(* IEC 61131-3 sources: AXOpen/src/components.keyence.vision/ctrl/src/Axo_IV3/TypesStructuresAndEnums, 15 files *)

(* ---- Axo_IV3_CommandControl.st ---- *)
NAMESPACE AXOpen.Components.Keyence.Vision
    {S7.extern=ReadWrite}
    {#ix-attr:[Container(Layout.Stack)]}
    CLASS PUBLIC Axo_IV3_CommandControl
        VAR PUBLIC
            {#ix-set:AttributeName = "<#Trigger request#>"}
            TriggerRequest                              : BOOL;                         //  QB0.0
            {#ix-set:AttributeName = "<#Master registration request#>"}
            MasterRegistrationRequest                   : BOOL;                         //  QB0.1
            {#ix-set:AttributeName = "<#Program switching request#>"}
            ProgramSwitchingRequest                     : BOOL;                         //  QB0.2
            {#ix-set:AttributeName = "<#Warning clear request#>"}
            WarningClearRequest                         : BOOL;                         //  QB0.3
            {#ix-set:AttributeName = "<#Statistics reset request#>"}
            StatisticsResetRequest                      : BOOL;                         //  QB0.4
            {#ix-set:AttributeName = "<#Buffer clear request#>"}
            BufferClearRequest                          : BOOL;                         //  QB0.5
            {#ix-set:AttributeName = "<#SD card saving stop request#>"}
            SdCardSavingStopRequest                     : BOOL;                         //  QB0.6
            {#ix-set:AttributeName = "<#Setting value change request#>"}
            SettingValueChangeRequest                   : BOOL;                         //  QB0.7
            {#ix-set:AttributeName = "<#Result acquisition complete notification#>"}
            ResultAcquisitionCompleteNotification       : BOOL;                         //  QB2.0
            {#ix-set:AttributeName = "<#Program number#>"}
            ProgramNo                                   : UINT;                         //  QW4
            {#ix-set:AttributeName = "<#Function 1: Limit set.no.(no OCR)/Master text set.no.(OCR)/FTP/SD-saved set.no.(FTP client/SD card saving function)#>"}
            Function_1                                  : WORD;                         //  QW6
            {#ix-set:AttributeName = "<#Function 2: Limit set.no.(no OCR)/Master text/number of letters(OCR)/FTP/SD-saving settings(FTP client/SD card saving function)#>"}
            Function_2                                  : DWORD;                        //  QD8
        END_VAR
    END_CLASS
END_NAMESPACE

(* ---- Axo_IV3_CommandStatusBits.st ---- *)
NAMESPACE AXOpen.Components.Keyence.Vision
    {S7.extern=ReadWrite}
    {#ix-attr:[Container(Layout.Wrap)]}
    CLASS PUBLIC Axo_IV3_CommandStatusBits
        VAR PUBLIC
            {#ix-attr:[Container(Layout.Stack)]}
            {#ix-attr:[Group(GroupLayout.GroupBox)]}
            {#ix-set:AttributeName = "<#Trigger response#>"}
            TriggerResponse : BOOL;                                                             // IB0.0
            {#ix-set:AttributeName = "<#Master registration response#>"}
            MasterRegistrationResponse : BOOL;                                                  // IB0.1
            {#ix-set:AttributeName = "<#Program switching response#>"}
            ProgramSwitchingResponse : BOOL;                                                    // IB0.2
            {#ix-set:AttributeName = "<#Warning clear response#>"}
            WarningClearResponse : BOOL;                                                        // IB0.3
            {#ix-set:AttributeName = "<#Statistics reset response#>"}
            StatisticsResetResponse : BOOL;                                                     // IB0.4
            {#ix-set:AttributeName = "<#Buffer clear response#>"}
            BufferClearResponse : BOOL;                                                         // IB0.5
            {#ix-set:AttributeName = "<#SD card saving stop response#>"}
            SdCardSavingStopResponse : BOOL;                                                    // IB0.6
            {#ix-set:AttributeName = "<#Setting value change response#>"}
            SettingValueChangeResponse : BOOL;                                                  // IB0.7

            {#ix-attr:[Container(Layout.Stack)]}
            {#ix-attr:[Group(GroupLayout.GroupBox)]}
            {#ix-set:AttributeName = "<#Trigger failed#>"}
            TriggerFailed : BOOL;                                                               // IB1.0
            {#ix-set:AttributeName = "<#Master registration failed#>"}
            MasterRegistrationFailed : BOOL;                                                    // IB1.1
            {#ix-set:AttributeName = "<#Program switching failed#>"}
            ProgramSwitchingFailed : BOOL;                                                      // IB1.2
                                                                                                // IB1.3
                                                                                                // IB1.4
                                                                                                // IB1.5
            {#ix-set:AttributeName = "<#SD card saving stop failed#>"}
            SdCardSavingStopFailed : BOOL;                                                      // IB1.6
            {#ix-set:AttributeName = "<#Setting value change failed#>"}
            SettingValueChangeFailed : BOOL;                                                    // IB1.7

            {#ix-attr:[Container(Layout.Stack)]}
            {#ix-attr:[Group(GroupLayout.GroupBox)]}
            {#ix-set:AttributeName = "<#Result available#>"}
            ResultAvailable : BOOL;                                                             // IB2.0
            {#ix-set:AttributeName = "<#Result update complete#>"}
            ResultUpdateComplete : BOOL;                                                        // IB2.1
            {#ix-set:AttributeName = "<#BUSY#>"}
            BUSY : BOOL;                                                                        // IB2.2
            {#ix-set:AttributeName = "<#Imaging status#>"}
            ImagingStatus : BOOL;                                                               // IB2.3
            {#ix-set:AttributeName = "<#RUN#>"}
            RUN : BOOL;                                                                         // IB2.4
            {#ix-set:AttributeName = "<#Ready#>"}
            Ready : BOOL;                                                                       // IB2.5
            {#ix-set:AttributeName = "<#Trigger ready#>"}
            TriggerReady : BOOL;                                                                // IB2.6
            {#ix-set:AttributeName = "<#SD card identification status#>"}
            SdCardIdentificationStatus : BOOL;                                                  // IB2.7

            {#ix-attr:[Container(Layout.Stack)]}
            {#ix-attr:[Group(GroupLayout.GroupBox)]}
            {#ix-set:AttributeName = "<#Sorting mode information#>"}
            SortingModeInformation : BOOL;                                                      // IB3.0
                                                                                                // IB3.1
                                                                                                // IB3.2
                                                                                                // IB3.3
            {#ix-set:AttributeName = "<#Insufficient free space on SD card#>"}
            InsufficientFreeSpaceOnSdCard : BOOL;                                               // IB3.4
            {#ix-set:AttributeName = "<#Buffer overrun#>"}
            BufferOverrun : BOOL;                                                               // IB3.5
            {#ix-set:AttributeName = "<#Warning#>"}
            Warning : BOOL;                                                                     // IB3.6
            {#ix-set:AttributeName = "<#Error#>"}
            Error : BOOL;                                                                       // IB3.7

        END_VAR
    END_CLASS
END_NAMESPACE

(* ---- Axo_IV3_Component_Status.st ---- *)
NAMESPACE AXOpen.Components.Keyence.Vision
    {S7.extern=ReadWrite}
    {#ix-attr:[Container(Layout.Stack)]}
    CLASS PUBLIC Axo_IV3_Component_Status EXTENDS AXOpen.Components.Abstractions.AxoComponent_Status
        VAR PUBLIC

        END_VAR
    END_CLASS
END_NAMESPACE

(* ---- Axo_IV3_Config.st ---- *)
NAMESPACE AXOpen.Components.Keyence.Vision
    {S7.extern=ReadWrite}
    {#ix-attr:[Container(Layout.Stack)]}
    CLASS PUBLIC Axo_IV3_Config
        VAR PUBLIC
            {#ix-set:AttributeName = "<#Info time#>"}
            InfoTime : LTIME := LT#5S;
            {#ix-set:AttributeName = "<#Error time#>"}
            ErrorTime : LTIME := LT#10S;
            {#ix-set:AttributeName = "<#Task timeout#>"}
            TaskTimeout : LTIME := LT#50S;
            {#ix-set:AttributeName = "<#Hardware IDs#>"}
            HWIDs : Axo_IV3_HWIDs;
        END_VAR
    END_CLASS
END_NAMESPACE

(* ---- Axo_IV3_Control.st ---- *)
NAMESPACE AXOpen.Components.Keyence.Vision
    {S7.extern=ReadWrite}
    {#ix-attr:[Container(Layout.Stack)]}
    CLASS PUBLIC Axo_IV3_Control
        VAR PUBLIC

        END_VAR
    END_CLASS
END_NAMESPACE

(* ---- Axo_IV3_DeviceResultBits_1.st ---- *)
NAMESPACE AXOpen.Components.Keyence.Vision
    {S7.extern=ReadWrite}
    {#ix-attr:[Container(Layout.Wrap)]}
    CLASS PUBLIC Axo_IV3_DeviceResultBits_1
        VAR PUBLIC
            {#ix-attr:[Container(Layout.Stack)]}
            {#ix-attr:[Group(GroupLayout.GroupBox)]}
            {#ix-set:AttributeName = "<#Overall judgment OK#>"}
            OverallJudgmentOK : BOOL;                                                           // IB4.0
            {#ix-set:AttributeName = "<#Position correction#>"}
            PositionCorrection : BOOL;                                                          // IB4.1
            {#ix-set:AttributeName = "<#LOGIC1#>"}
            LOGIC1 : BOOL;                                                                      // IB4.2
            {#ix-set:AttributeName = "<#LOGIC2#>"}
            LOGIC2 : BOOL;                                                                      // IB4.3
            {#ix-set:AttributeName = "<#LOGIC3#>"}
            LOGIC3 : BOOL;                                                                      // IB4.4
            {#ix-set:AttributeName = "<#LOGIC4#>"}
            LOGIC4 : BOOL;                                                                      // IB4.5
            {#ix-set:AttributeName = "<#Overall judgment NG#>"}
            OverallJudgmentNG : BOOL;                                                           // IB4.6
                                                                                                // IB4.7
            {#ix-attr:[Container(Layout.Stack)]}
            {#ix-attr:[Group(GroupLayout.GroupBox)]}
            {#ix-set:AttributeName = "<#Tool 1#>"}
            Tool_1 : BOOL;                                                                      // IB6.0
            {#ix-set:AttributeName = "<#Tool 2#>"}
            Tool_2 : BOOL;                                                                      // IB6.1
            {#ix-set:AttributeName = "<#Tool 3#>"}
            Tool_3 : BOOL;                                                                      // IB6.2
            {#ix-set:AttributeName = "<#Tool 4#>"}
            Tool_4 : BOOL;                                                                      // IB6.3
            {#ix-set:AttributeName = "<#Tool 5#>"}
            Tool_5 : BOOL;                                                                      // IB6.4
            {#ix-set:AttributeName = "<#Tool 6#>"}
            Tool_6 : BOOL;                                                                      // IB6.5
            {#ix-set:AttributeName = "<#Tool 7#>"}
            Tool_7 : BOOL;                                                                      // IB6.6
            {#ix-set:AttributeName = "<#Tool 8#>"}
            Tool_8 : BOOL;                                                                      // IB6.7
            {#ix-set:AttributeName = "<#Tool 9#>"}
            Tool_9 : BOOL;                                                                      // IB7.0
            {#ix-set:AttributeName = "<#Tool 10#>"}
            Tool_10 : BOOL;                                                                     // IB7.1
            {#ix-set:AttributeName = "<#Tool 11#>"}
            Tool_11 : BOOL;                                                                     // IB7.2
            {#ix-set:AttributeName = "<#Tool 12#>"}
            Tool_12 : BOOL;                                                                     // IB7.3
            {#ix-set:AttributeName = "<#Tool 13#>"}
            Tool_13 : BOOL;                                                                     // IB7.4
            {#ix-set:AttributeName = "<#Tool 14#>"}
            Tool_14 : BOOL;                                                                     // IB7.5
            {#ix-set:AttributeName = "<#Tool 15#>"}
            Tool_15 : BOOL;                                                                     // IB7.6
            {#ix-set:AttributeName = "<#Tool 16#>"}
            Tool_16 : BOOL;                                                                     // IB7.7
        END_VAR
    END_CLASS
END_NAMESPACE

(* ---- Axo_IV3_DeviceResultBits_2.st ---- *)
NAMESPACE AXOpen.Components.Keyence.Vision
    {S7.extern=ReadWrite}
    {#ix-attr:[Container(Layout.Wrap)]}
    CLASS PUBLIC Axo_IV3_DeviceResultBits_2
        VAR PUBLIC
            {#ix-attr:[Container(Layout.Stack)]}
            {#ix-attr:[Group(GroupLayout.GroupBox)]}
            {#ix-set:AttributeName = "<#Master number/total status product type#>"}
            MasterNumber : UINT;                                                                // IW1352

            {#ix-attr:[Container(Layout.Stack)]}
            {#ix-attr:[Group(GroupLayout.GroupBox)]}
            {#ix-set:AttributeName = "<#Tool 17#>"}
            Tool_17 : BOOL;                                                                      // IB1354.0
            {#ix-set:AttributeName = "<#Tool 18#>"}
            Tool_18 : BOOL;                                                                      // IB1354.1
            {#ix-set:AttributeName = "<#Tool 19#>"}
            Tool_19 : BOOL;                                                                      // IB1354.2
            {#ix-set:AttributeName = "<#Tool 20#>"}
            Tool_20 : BOOL;                                                                      // IB1354.3
            {#ix-set:AttributeName = "<#Tool 21#>"}
            Tool_21 : BOOL;                                                                      // IB1354.4
            {#ix-set:AttributeName = "<#Tool 22#>"}
            Tool_22 : BOOL;                                                                      // IB1354.5
            {#ix-set:AttributeName = "<#Tool 23#>"}
            Tool_23 : BOOL;                                                                      // IB1354.6
            {#ix-set:AttributeName = "<#Tool 24#>"}
            Tool_24 : BOOL;                                                                      // IB1354.7
            {#ix-set:AttributeName = "<#Tool 25#>"}
            Tool_25 : BOOL;                                                                      // IB1355.0
            {#ix-set:AttributeName = "<#Tool 26#>"}
            Tool_26 : BOOL;                                                                      // IB1355.1
            {#ix-set:AttributeName = "<#Tool 27#>"}
            Tool_27 : BOOL;                                                                      // IB1355.2
            {#ix-set:AttributeName = "<#Tool 28#>"}
            Tool_28 : BOOL;                                                                      // IB1355.3
            {#ix-set:AttributeName = "<#Tool 29#>"}
            Tool_29 : BOOL;                                                                      // IB1355.4
            {#ix-set:AttributeName = "<#Tool 30#>"}
            Tool_30 : BOOL;                                                                      // IB1355.5
            {#ix-set:AttributeName = "<#Tool 31#>"}
            Tool_31 : BOOL;                                                                      // IB1355.6
            {#ix-set:AttributeName = "<#Tool 32#>"}
            Tool_32 : BOOL;                                                                      // IB1355.7
            {#ix-set:AttributeName = "<#Tool 33#>"}
            Tool_33 : BOOL;                                                                      // IB1356.0
            {#ix-set:AttributeName = "<#Tool 34#>"}
            Tool_34 : BOOL;                                                                      // IB1356.1
            {#ix-set:AttributeName = "<#Tool 35#>"}
            Tool_35 : BOOL;                                                                      // IB1356.2
            {#ix-set:AttributeName = "<#Tool 36#>"}
            Tool_36 : BOOL;                                                                      // IB1356.3
            {#ix-set:AttributeName = "<#Tool 37#>"}
            Tool_37 : BOOL;                                                                      // IB1356.4
            {#ix-set:AttributeName = "<#Tool 38#>"}
            Tool_38 : BOOL;                                                                      // IB1356.5
            {#ix-set:AttributeName = "<#Tool 39#>"}
            Tool_39 : BOOL;                                                                      // IB1356.6
            {#ix-set:AttributeName = "<#Tool 40#>"}
            Tool_40 : BOOL;                                                                      // IB1356.7
            {#ix-set:AttributeName = "<#Tool 41#>"}
            Tool_41 : BOOL;                                                                      // IB1357.0
            {#ix-set:AttributeName = "<#Tool 42#>"}
            Tool_42 : BOOL;                                                                      // IB1357.1
            {#ix-set:AttributeName = "<#Tool 43#>"}
            Tool_43 : BOOL;                                                                      // IB1357.2
            {#ix-set:AttributeName = "<#Tool 44#>"}
            Tool_44 : BOOL;                                                                      // IB1357.3
            {#ix-set:AttributeName = "<#Tool 45#>"}
            Tool_45 : BOOL;                                                                      // IB1357.4
            {#ix-set:AttributeName = "<#Tool 46#>"}
            Tool_46 : BOOL;                                                                      // IB1357.5
            {#ix-set:AttributeName = "<#Tool 47#>"}
            Tool_47 : BOOL;                                                                      // IB1357.6
            {#ix-set:AttributeName = "<#Tool 48#>"}
            Tool_48 : BOOL;                                                                      // IB1357.7
            {#ix-set:AttributeName = "<#Tool 49#>"}
            Tool_49 : BOOL;                                                                      // IB1358.0
            {#ix-set:AttributeName = "<#Tool 50#>"}
            Tool_50 : BOOL;                                                                      // IB1358.1
            {#ix-set:AttributeName = "<#Tool 51#>"}
            Tool_51 : BOOL;                                                                      // IB1358.2
            {#ix-set:AttributeName = "<#Tool 52#>"}
            Tool_52 : BOOL;                                                                      // IB1358.3
            {#ix-set:AttributeName = "<#Tool 53#>"}
            Tool_53 : BOOL;                                                                      // IB1358.4
            {#ix-set:AttributeName = "<#Tool 54#>"}
            Tool_54 : BOOL;                                                                      // IB1358.5
            {#ix-set:AttributeName = "<#Tool 55#>"}
            Tool_55 : BOOL;                                                                      // IB1358.6
            {#ix-set:AttributeName = "<#Tool 56#>"}
            Tool_56 : BOOL;                                                                      // IB1358.7
            {#ix-set:AttributeName = "<#Tool 57#>"}
            Tool_57 : BOOL;                                                                      // IB1359.0
            {#ix-set:AttributeName = "<#Tool 58#>"}
            Tool_58 : BOOL;                                                                      // IB1359.1
            {#ix-set:AttributeName = "<#Tool 59#>"}
            Tool_59 : BOOL;                                                                      // IB1359.2
            {#ix-set:AttributeName = "<#Tool 60#>"}
            Tool_60 : BOOL;                                                                      // IB1359.3
            {#ix-set:AttributeName = "<#Tool 61#>"}
            Tool_61 : BOOL;                                                                      // IB1359.4
            {#ix-set:AttributeName = "<#Tool 62#>"}
            Tool_62 : BOOL;                                                                      // IB1359.5
            {#ix-set:AttributeName = "<#Tool 63#>"}
            Tool_63 : BOOL;                                                                      // IB1359.6
            {#ix-set:AttributeName = "<#Tool 64#>"}
            Tool_64 : BOOL;                                                                      // IB1359.7
        END_VAR
    END_CLASS
END_NAMESPACE

(* ---- Axo_IV3_DeviceStatistics.st ---- *)
NAMESPACE AXOpen.Components.Keyence.Vision
    {S7.extern=ReadWrite}
    {#ix-attr:[Container(Layout.Wrap)]}
    CLASS PUBLIC Axo_IV3_DeviceStatistics
        VAR PUBLIC
            {#ix-attr:[Container(Layout.Stack)]}
            {#ix-attr:[Group(GroupLayout.GroupBox)]}
            {#ix-set:AttributeName = "<#Processing time MAX#>"}
            ProcessingTimeMax : UINT;                                                           // IW24
            {#ix-set:AttributeName = "<#Processing time MIN#>"}
            ProcessingTimeMin : UINT;                                                           // IW26
            {#ix-set:AttributeName = "<#Processing time AVE#>"}
            ProcessingTimeAve : UINT;                                                           // IW28
                                                                                                // IW30
            {#ix-set:AttributeName = "<#Number of triggers#>"}
            NumberOfTriggers : UDINT;                                                           // ID32
            {#ix-set:AttributeName = "<#Number of OKs#>"}
            NumberOfOKs : UDINT;                                                                // ID36
            {#ix-set:AttributeName = "<#Number of NGs#>"}
            NumberOfNGs : UDINT;                                                                // ID40
            {#ix-set:AttributeName = "<#Number of trigger errors#>"}
            NumberOfTriggerErrors : UDINT;                                                      // ID44
                                                                                                // ID48
        END_VAR
    END_CLASS
END_NAMESPACE

(* ---- Axo_IV3_DeviceStatusWords.st ---- *)
NAMESPACE AXOpen.Components.Keyence.Vision
    {S7.extern=ReadWrite}
    {#ix-attr:[Container(Layout.Wrap)]}
    CLASS PUBLIC Axo_IV3_DeviceStatusWords
        VAR PUBLIC
            {#ix-attr:[Container(Layout.Stack)]}
            {#ix-attr:[Group(GroupLayout.GroupBox)]}
            {#ix-set:AttributeName = "<#Error No.#>"}
            ErrorNo : UINT;                                                                     // IW8
            {#ix-set:AttributeName = "<#Warning No.#>"}
            WarningNo : UINT;                                                                   // IW10
            {#ix-set:AttributeName = "<#Number of remaining buffers#>"}
            NumberOfRemainingBuffers : UINT;                                                    // IW12
            {#ix-set:AttributeName = "<#Checksum#>"}
            Checksum : UINT;                                                                    // IW14
            {#ix-set:AttributeName = "<#Current program No.#>"}
            CurrentProgramNo : UINT;                                                            // IW16
            {#ix-set:AttributeName = "<#Program No. during judgment#>"}
            ProgramNoDuringJudgment : UINT;                                                     // IW18
            {#ix-set:AttributeName = "<#Result No.#>"}
            ResultNo : UINT;                                                                    // IW20
            {#ix-set:AttributeName = "<#Processing time#>"}
            ProcessingTime : UINT;                                                              // IW22
        END_VAR
    END_CLASS
END_NAMESPACE

(* ---- Axo_IV3_HWIDs.st ---- *)
NAMESPACE AXOpen.Components.Keyence.Vision
   {S7.extern=ReadWrite}
	CLASS Axo_IV3_HWIDs
      VAR PUBLIC
         {#ix-set:AttributeName = "<#Hardware ID  of the device#>"}
         HW_Device              :  UINT;
         {#ix-set:AttributeName = "<#Hardware ID of the 'CommandControl' submodule#>"}
         HwID_CommandControl            :   UINT;
         {#ix-set:AttributeName = "<#Hardware ID of the 'CommandStatusBits' submodule#>"}
         HwID_CommandStatusBits            :   UINT;
         {#ix-set:AttributeName = "<#Hardware ID of the 'DeviceResultBits_1' submodule#>"}
         HwID_DeviceResultBits_1            :   UINT;
         {#ix-set:AttributeName = "<#Hardware ID of the 'DeviceStatusWords' submodule#>"}
         HwID_DeviceStatusWords            :   UINT;
         {#ix-set:AttributeName = "<#Hardware ID of the 'DeviceStatistics' submodule#>"}
         HwID_DeviceStatistics            :   UINT;
         {#ix-set:AttributeName = "<#Hardware ID of the 'PositionAdjustResult' submodule#>"}
         HwID_PositionAdjustResult            :   UINT;
         {#ix-set:AttributeName = "<#Hardware ID of the 'ToolResult_1' submodule#>"}
         HwID_ToolResult_1            :   UINT;
         {#ix-set:AttributeName = "<#Hardware ID of the 'ToolResult_2' submodule#>"}
         HwID_ToolResult_2            :   UINT;
         {#ix-set:AttributeName = "<#Hardware ID of the 'ToolResult_3' submodule#>"}
         HwID_ToolResult_3            :   UINT;
         {#ix-set:AttributeName = "<#Hardware ID of the 'ToolResult_4' submodule#>"}
         HwID_ToolResult_4            :   UINT;
         {#ix-set:AttributeName = "<#Hardware ID of the 'ToolResult_5' submodule#>"}
         HwID_ToolResult_5            :   UINT;
         {#ix-set:AttributeName = "<#Hardware ID of the 'ToolResult_6' submodule#>"}
         HwID_ToolResult_6            :   UINT;
         {#ix-set:AttributeName = "<#Hardware ID of the 'ToolResult_7' submodule#>"}
         HwID_ToolResult_7            :   UINT;
         {#ix-set:AttributeName = "<#Hardware ID of the 'ToolResult_8' submodule#>"}
         HwID_ToolResult_8            :   UINT;
         {#ix-set:AttributeName = "<#Hardware ID of the 'ToolResult_9' submodule#>"}
         HwID_ToolResult_9            :   UINT;
         {#ix-set:AttributeName = "<#Hardware ID of the 'ToolResult_10' submodule#>"}
         HwID_ToolResult_10            :   UINT;
         {#ix-set:AttributeName = "<#Hardware ID of the 'ToolResult_11' submodule#>"}
         HwID_ToolResult_11            :   UINT;
         {#ix-set:AttributeName = "<#Hardware ID of the 'ToolResult_12' submodule#>"}
         HwID_ToolResult_12            :   UINT;
         {#ix-set:AttributeName = "<#Hardware ID of the 'ToolResult_13' submodule#>"}
         HwID_ToolResult_13            :   UINT;
         {#ix-set:AttributeName = "<#Hardware ID of the 'ToolResult_14' submodule#>"}
         HwID_ToolResult_14            :   UINT;
         {#ix-set:AttributeName = "<#Hardware ID of the 'ToolResult_15' submodule#>"}
         HwID_ToolResult_15            :   UINT;
         {#ix-set:AttributeName = "<#Hardware ID of the 'ToolResult_16' submodule#>"}
         HwID_ToolResult_16            :   UINT;
         {#ix-set:AttributeName = "<#Hardware ID of the 'ToolResult_17' submodule#>"}
         HwID_ToolResult_17            :   UINT;
         {#ix-set:AttributeName = "<#Hardware ID of the 'ToolResult_18' submodule#>"}
         HwID_ToolResult_18            :   UINT;
         {#ix-set:AttributeName = "<#Hardware ID of the 'ToolResult_19' submodule#>"}
         HwID_ToolResult_19            :   UINT;
         {#ix-set:AttributeName = "<#Hardware ID of the 'ToolResult_20' submodule#>"}
         HwID_ToolResult_20            :   UINT;
         {#ix-set:AttributeName = "<#Hardware ID of the 'ToolResult_21' submodule#>"}
         HwID_ToolResult_21            :   UINT;
         {#ix-set:AttributeName = "<#Hardware ID of the 'ToolResult_22' submodule#>"}
         HwID_ToolResult_22            :   UINT;
         {#ix-set:AttributeName = "<#Hardware ID of the 'ToolResult_23' submodule#>"}
         HwID_ToolResult_23            :   UINT;
         {#ix-set:AttributeName = "<#Hardware ID of the 'ToolResult_24' submodule#>"}
         HwID_ToolResult_24            :   UINT;
         {#ix-set:AttributeName = "<#Hardware ID of the 'ToolResult_25' submodule#>"}
         HwID_ToolResult_25            :   UINT;
         {#ix-set:AttributeName = "<#Hardware ID of the 'ToolResult_26' submodule#>"}
         HwID_ToolResult_26            :   UINT;
         {#ix-set:AttributeName = "<#Hardware ID of the 'ToolResult_27' submodule#>"}
         HwID_ToolResult_27            :   UINT;
         {#ix-set:AttributeName = "<#Hardware ID of the 'ToolResult_28' submodule#>"}
         HwID_ToolResult_28            :   UINT;
         {#ix-set:AttributeName = "<#Hardware ID of the 'ToolResult_29' submodule#>"}
         HwID_ToolResult_29            :   UINT;
         {#ix-set:AttributeName = "<#Hardware ID of the 'ToolResult_30' submodule#>"}
         HwID_ToolResult_30            :   UINT;
         {#ix-set:AttributeName = "<#Hardware ID of the 'ToolResult_31' submodule#>"}
         HwID_ToolResult_31            :   UINT;
         {#ix-set:AttributeName = "<#Hardware ID of the 'ToolResult_32' submodule#>"}
         HwID_ToolResult_32            :   UINT;
         {#ix-set:AttributeName = "<#Hardware ID of the 'ToolResult_33' submodule#>"}
         HwID_ToolResult_33            :   UINT;
         {#ix-set:AttributeName = "<#Hardware ID of the 'ToolResult_34' submodule#>"}
         HwID_ToolResult_34            :   UINT;
         {#ix-set:AttributeName = "<#Hardware ID of the 'ToolResult_35' submodule#>"}
         HwID_ToolResult_35            :   UINT;
         {#ix-set:AttributeName = "<#Hardware ID of the 'ToolResult_36' submodule#>"}
         HwID_ToolResult_36            :   UINT;
         {#ix-set:AttributeName = "<#Hardware ID of the 'ToolResult_37' submodule#>"}
         HwID_ToolResult_37            :   UINT;
         {#ix-set:AttributeName = "<#Hardware ID of the 'ToolResult_38' submodule#>"}
         HwID_ToolResult_38            :   UINT;
         {#ix-set:AttributeName = "<#Hardware ID of the 'ToolResult_39' submodule#>"}
         HwID_ToolResult_39            :   UINT;
         {#ix-set:AttributeName = "<#Hardware ID of the 'ToolResult_40' submodule#>"}
         HwID_ToolResult_40            :   UINT;
         {#ix-set:AttributeName = "<#Hardware ID of the 'ToolResult_41' submodule#>"}
         HwID_ToolResult_41            :   UINT;
         {#ix-set:AttributeName = "<#Hardware ID of the 'ToolResult_42' submodule#>"}
         HwID_ToolResult_42            :   UINT;
         {#ix-set:AttributeName = "<#Hardware ID of the 'ToolResult_43' submodule#>"}
         HwID_ToolResult_43            :   UINT;
         {#ix-set:AttributeName = "<#Hardware ID of the 'ToolResult_44' submodule#>"}
         HwID_ToolResult_44            :   UINT;
         {#ix-set:AttributeName = "<#Hardware ID of the 'ToolResult_45' submodule#>"}
         HwID_ToolResult_45            :   UINT;
         {#ix-set:AttributeName = "<#Hardware ID of the 'ToolResult_46' submodule#>"}
         HwID_ToolResult_46            :   UINT;
         {#ix-set:AttributeName = "<#Hardware ID of the 'ToolResult_47' submodule#>"}
         HwID_ToolResult_47            :   UINT;
         {#ix-set:AttributeName = "<#Hardware ID of the 'ToolResult_48' submodule#>"}
         HwID_ToolResult_48            :   UINT;
         {#ix-set:AttributeName = "<#Hardware ID of the 'ToolResult_49' submodule#>"}
         HwID_ToolResult_49            :   UINT;
         {#ix-set:AttributeName = "<#Hardware ID of the 'ToolResult_50' submodule#>"}
         HwID_ToolResult_50            :   UINT;
         {#ix-set:AttributeName = "<#Hardware ID of the 'ToolResult_51' submodule#>"}
         HwID_ToolResult_51            :   UINT;
         {#ix-set:AttributeName = "<#Hardware ID of the 'ToolResult_52' submodule#>"}
         HwID_ToolResult_52            :   UINT;
         {#ix-set:AttributeName = "<#Hardware ID of the 'ToolResult_53' submodule#>"}
         HwID_ToolResult_53            :   UINT;
         {#ix-set:AttributeName = "<#Hardware ID of the 'ToolResult_54' submodule#>"}
         HwID_ToolResult_54            :   UINT;
         {#ix-set:AttributeName = "<#Hardware ID of the 'ToolResult_55' submodule#>"}
         HwID_ToolResult_55            :   UINT;
         {#ix-set:AttributeName = "<#Hardware ID of the 'ToolResult_56' submodule#>"}
         HwID_ToolResult_56            :   UINT;
         {#ix-set:AttributeName = "<#Hardware ID of the 'ToolResult_57' submodule#>"}
         HwID_ToolResult_57            :   UINT;
         {#ix-set:AttributeName = "<#Hardware ID of the 'ToolResult_58' submodule#>"}
         HwID_ToolResult_58            :   UINT;
         {#ix-set:AttributeName = "<#Hardware ID of the 'ToolResult_59' submodule#>"}
         HwID_ToolResult_59            :   UINT;
         {#ix-set:AttributeName = "<#Hardware ID of the 'ToolResult_60' submodule#>"}
         HwID_ToolResult_60            :   UINT;
         {#ix-set:AttributeName = "<#Hardware ID of the 'ToolResult_61' submodule#>"}
         HwID_ToolResult_61            :   UINT;
         {#ix-set:AttributeName = "<#Hardware ID of the 'ToolResult_62' submodule#>"}
         HwID_ToolResult_62            :   UINT;
         {#ix-set:AttributeName = "<#Hardware ID of the 'ToolResult_63' submodule#>"}
         HwID_ToolResult_63            :   UINT;
         {#ix-set:AttributeName = "<#Hardware ID of the 'ToolResult_64' submodule#>"}
         HwID_ToolResult_64            :   UINT;
         {#ix-set:AttributeName = "<#Hardware ID of the 'DeviceResultBits_2' submodule#>"}
         HwID_DeviceResultBits_2            :   UINT;
      END_VAR
   END_CLASS
END_NAMESPACE

(* ---- Axo_IV3_In.st ---- *)
NAMESPACE AXOpen.Components.Keyence.Vision
    {S7.extern=ReadWrite}
    {#ix-attr:[Container(Layout.Wrap)]}
    CLASS PUBLIC Axo_IV3_In
        VAR PUBLIC
            // {#ix-set:AttributeName = "<#Status#>"}
            // {#ix-attr:[ReadOnly()]}
            // Status           :   Axo_IV3_Status;
            {#ix-attr:[Container(Layout.Stack)]}
            {#ix-attr:[Group(GroupLayout.GroupBox)]}
            {#ix-set:AttributeName = "<#Command status bits#>"}
            {#ix-attr:[ReadOnly()]}
            CommandStatusBits           :   Axo_IV3_CommandStatusBits;                              // IB0-IB3

            {#ix-attr:[Container(Layout.Stack)]}
            {#ix-attr:[Group(GroupLayout.GroupBox)]}
            {#ix-set:AttributeName = "<#Device result bits 1#>"}
            {#ix-attr:[ReadOnly()]}
            DeviceResultBits_1          :   Axo_IV3_DeviceResultBits_1;                             // IB4-IB7

            {#ix-attr:[Container(Layout.Stack)]}
            {#ix-attr:[Group(GroupLayout.GroupBox)]}
            {#ix-set:AttributeName = "<#Device status words#>"}
            {#ix-attr:[ReadOnly()]}
            DeviceStatusWords           :   Axo_IV3_DeviceStatusWords;                              // IB8-IB23

            {#ix-attr:[Container(Layout.Stack)]}
            {#ix-attr:[Group(GroupLayout.GroupBox)]}
            {#ix-set:AttributeName = "<#Device statistics#>"}
            {#ix-attr:[ReadOnly()]}
            DeviceStatistics            :   Axo_IV3_DeviceStatistics;                               // IB24-IB51

            {#ix-attr:[Container(Layout.Stack)]}
            {#ix-attr:[Group(GroupLayout.GroupBox)]}
            {#ix-set:AttributeName = "<#Position adjust result#>"}
            {#ix-attr:[ReadOnly()]}
            PositionAdjustResult        :   Axo_IV3_PositionAdjustResult;                           // IB52-IB71

            {#ix-attr:[Container(Layout.Stack)]}
            {#ix-attr:[Group(GroupLayout.GroupBox)]}
            {#ix-set:AttributeName = "<#Tool result 1#>"}
            ToolResult_1 : Axo_IV3_ToolResult;                                                      // IB72-IB91
            {#ix-attr:[Container(Layout.Stack)]}
            {#ix-attr:[Group(GroupLayout.GroupBox)]}
            {#ix-set:AttributeName = "<#Tool result 2#>"}
            ToolResult_2 : Axo_IV3_ToolResult;                                                      // IB92-IB111
            {#ix-attr:[Container(Layout.Stack)]}
            {#ix-attr:[Group(GroupLayout.GroupBox)]}
            {#ix-set:AttributeName = "<#Tool result 3#>"}
            ToolResult_3 : Axo_IV3_ToolResult;                                                      // IB112-IB131
            {#ix-attr:[Container(Layout.Stack)]}
            {#ix-attr:[Group(GroupLayout.GroupBox)]}
            {#ix-set:AttributeName = "<#Tool result 4#>"}
            ToolResult_4 : Axo_IV3_ToolResult;                                                      // IB132-IB151
            {#ix-attr:[Container(Layout.Stack)]}
            {#ix-attr:[Group(GroupLayout.GroupBox)]}
            {#ix-set:AttributeName = "<#Tool result 5#>"}
            ToolResult_5 : Axo_IV3_ToolResult;                                                      // IB152-IB171
            {#ix-attr:[Container(Layout.Stack)]}
            {#ix-attr:[Group(GroupLayout.GroupBox)]}
            {#ix-set:AttributeName = "<#Tool result 6#>"}
            ToolResult_6 : Axo_IV3_ToolResult;                                                      // IB172-IB191
            {#ix-attr:[Container(Layout.Stack)]}
            {#ix-attr:[Group(GroupLayout.GroupBox)]}
            {#ix-set:AttributeName = "<#Tool result 7#>"}
            ToolResult_7 : Axo_IV3_ToolResult;                                                      // IB192-IB211
            {#ix-attr:[Container(Layout.Stack)]}
            {#ix-attr:[Group(GroupLayout.GroupBox)]}
            {#ix-set:AttributeName = "<#Tool result 8#>"}
            ToolResult_8 : Axo_IV3_ToolResult;                                                      // IB212-IB231
            {#ix-attr:[Container(Layout.Stack)]}
            {#ix-attr:[Group(GroupLayout.GroupBox)]}
            {#ix-set:AttributeName = "<#Tool result 9#>"}
            ToolResult_9 : Axo_IV3_ToolResult;                                                      // IB232-IB251
            {#ix-attr:[Container(Layout.Stack)]}
            {#ix-attr:[Group(GroupLayout.GroupBox)]}
            {#ix-set:AttributeName = "<#Tool result 10#>"}
            ToolResult_10 : Axo_IV3_ToolResult;                                                     // IB252-IB271
            {#ix-attr:[Container(Layout.Stack)]}
            {#ix-attr:[Group(GroupLayout.GroupBox)]}
            {#ix-set:AttributeName = "<#Tool result 11#>"}
            ToolResult_11 : Axo_IV3_ToolResult;                                                     // IB272-IB291
            {#ix-attr:[Container(Layout.Stack)]}
            {#ix-attr:[Group(GroupLayout.GroupBox)]}
            {#ix-set:AttributeName = "<#Tool result 12#>"}
            ToolResult_12 : Axo_IV3_ToolResult;                                                     // IB292-IB311
            {#ix-attr:[Container(Layout.Stack)]}
            {#ix-attr:[Group(GroupLayout.GroupBox)]}
            {#ix-set:AttributeName = "<#Tool result 13#>"}
            ToolResult_13 : Axo_IV3_ToolResult;                                                     // IB312-IB331
            {#ix-attr:[Container(Layout.Stack)]}
            {#ix-attr:[Group(GroupLayout.GroupBox)]}
            {#ix-set:AttributeName = "<#Tool result 14#>"}
            ToolResult_14 : Axo_IV3_ToolResult;                                                     // IB332-IB351
            {#ix-attr:[Container(Layout.Stack)]}
            {#ix-attr:[Group(GroupLayout.GroupBox)]}
            {#ix-set:AttributeName = "<#Tool result 15#>"}
            ToolResult_15 : Axo_IV3_ToolResult;                                                     // IB352-IB371
            {#ix-attr:[Container(Layout.Stack)]}
            {#ix-attr:[Group(GroupLayout.GroupBox)]}
            {#ix-set:AttributeName = "<#Tool result 16#>"}
            ToolResult_16 : Axo_IV3_ToolResult;                                                     // IB372-IB391
            {#ix-attr:[Container(Layout.Stack)]}
            {#ix-attr:[Group(GroupLayout.GroupBox)]}
            {#ix-set:AttributeName = "<#Tool result 17#>"}
            ToolResult_17 : Axo_IV3_ToolResult;                                                     // IB392-IB411
            {#ix-attr:[Container(Layout.Stack)]}
            {#ix-attr:[Group(GroupLayout.GroupBox)]}
            {#ix-set:AttributeName = "<#Tool result 18#>"}
            ToolResult_18 : Axo_IV3_ToolResult;                                                     // IB412-IB431
            {#ix-attr:[Container(Layout.Stack)]}
            {#ix-attr:[Group(GroupLayout.GroupBox)]}
            {#ix-set:AttributeName = "<#Tool result 19#>"}
            ToolResult_19 : Axo_IV3_ToolResult;                                                     // IB432-IB451
            {#ix-attr:[Container(Layout.Stack)]}
            {#ix-attr:[Group(GroupLayout.GroupBox)]}
            {#ix-set:AttributeName = "<#Tool result 20#>"}
            ToolResult_20 : Axo_IV3_ToolResult;                                                     // IB452-IB471
            {#ix-attr:[Container(Layout.Stack)]}
            {#ix-attr:[Group(GroupLayout.GroupBox)]}
            {#ix-set:AttributeName = "<#Tool result 21#>"}
            ToolResult_21 : Axo_IV3_ToolResult;                                                     // IB472-IB491
            {#ix-attr:[Container(Layout.Stack)]}
            {#ix-attr:[Group(GroupLayout.GroupBox)]}
            {#ix-set:AttributeName = "<#Tool result 22#>"}
            ToolResult_22 : Axo_IV3_ToolResult;                                                     // IB492-IB511
            {#ix-attr:[Container(Layout.Stack)]}
            {#ix-attr:[Group(GroupLayout.GroupBox)]}
            {#ix-set:AttributeName = "<#Tool result 23#>"}
            ToolResult_23 : Axo_IV3_ToolResult;                                                     // IB512-IB531
            {#ix-attr:[Container(Layout.Stack)]}
            {#ix-attr:[Group(GroupLayout.GroupBox)]}
            {#ix-set:AttributeName = "<#Tool result 24#>"}
            ToolResult_24 : Axo_IV3_ToolResult;                                                     // IB532-IB551
            {#ix-attr:[Container(Layout.Stack)]}
            {#ix-attr:[Group(GroupLayout.GroupBox)]}
            {#ix-set:AttributeName = "<#Tool result 25#>"}
            ToolResult_25 : Axo_IV3_ToolResult;                                                     // IB552-IB571
            {#ix-attr:[Container(Layout.Stack)]}
            {#ix-attr:[Group(GroupLayout.GroupBox)]}
            {#ix-set:AttributeName = "<#Tool result 26#>"}
            ToolResult_26 : Axo_IV3_ToolResult;                                                     // IB572-IB591
            {#ix-attr:[Container(Layout.Stack)]}
            {#ix-attr:[Group(GroupLayout.GroupBox)]}
            {#ix-set:AttributeName = "<#Tool result 27#>"}
            ToolResult_27 : Axo_IV3_ToolResult;                                                     // IB592-IB611
            {#ix-attr:[Container(Layout.Stack)]}
            {#ix-attr:[Group(GroupLayout.GroupBox)]}
            {#ix-set:AttributeName = "<#Tool result 28#>"}
            ToolResult_28 : Axo_IV3_ToolResult;                                                     // IB612-IB631
            {#ix-attr:[Container(Layout.Stack)]}
            {#ix-attr:[Group(GroupLayout.GroupBox)]}
            {#ix-set:AttributeName = "<#Tool result 29#>"}
            ToolResult_29 : Axo_IV3_ToolResult;                                                     // IB632-IB651
            {#ix-attr:[Container(Layout.Stack)]}
            {#ix-attr:[Group(GroupLayout.GroupBox)]}
            {#ix-set:AttributeName = "<#Tool result 30#>"}
            ToolResult_30 : Axo_IV3_ToolResult;                                                     // IB652-IB671
            {#ix-attr:[Container(Layout.Stack)]}
            {#ix-attr:[Group(GroupLayout.GroupBox)]}
            {#ix-set:AttributeName = "<#Tool result 31#>"}
            ToolResult_31 : Axo_IV3_ToolResult;                                                     // IB672-IB691
            {#ix-attr:[Container(Layout.Stack)]}
            {#ix-attr:[Group(GroupLayout.GroupBox)]}
            {#ix-set:AttributeName = "<#Tool result 32#>"}
            ToolResult_32 : Axo_IV3_ToolResult;                                                     // IB692-IB711
            {#ix-attr:[Container(Layout.Stack)]}
            {#ix-attr:[Group(GroupLayout.GroupBox)]}
            {#ix-set:AttributeName = "<#Tool result 33#>"}
            ToolResult_33 : Axo_IV3_ToolResult;                                                     // IB712-IB731
            {#ix-attr:[Container(Layout.Stack)]}
            {#ix-attr:[Group(GroupLayout.GroupBox)]}
            {#ix-set:AttributeName = "<#Tool result 34#>"}
            ToolResult_34 : Axo_IV3_ToolResult;                                                     // IB732-IB751
            {#ix-attr:[Container(Layout.Stack)]}
            {#ix-attr:[Group(GroupLayout.GroupBox)]}
            {#ix-set:AttributeName = "<#Tool result 35#>"}
            ToolResult_35 : Axo_IV3_ToolResult;                                                     // IB752-IB771
            {#ix-attr:[Container(Layout.Stack)]}
            {#ix-attr:[Group(GroupLayout.GroupBox)]}
            {#ix-set:AttributeName = "<#Tool result 36#>"}
            ToolResult_36 : Axo_IV3_ToolResult;                                                     // IB772-IB791
            {#ix-attr:[Container(Layout.Stack)]}
            {#ix-attr:[Group(GroupLayout.GroupBox)]}
            {#ix-set:AttributeName = "<#Tool result 37#>"}
            ToolResult_37 : Axo_IV3_ToolResult;                                                     // IB792-IB811
            {#ix-attr:[Container(Layout.Stack)]}
            {#ix-attr:[Group(GroupLayout.GroupBox)]}
            {#ix-set:AttributeName = "<#Tool result 38#>"}
            ToolResult_38 : Axo_IV3_ToolResult;                                                     // IB812-IB831
            {#ix-attr:[Container(Layout.Stack)]}
            {#ix-attr:[Group(GroupLayout.GroupBox)]}
            {#ix-set:AttributeName = "<#Tool result 39#>"}
            ToolResult_39 : Axo_IV3_ToolResult;                                                     // IB832-IB851
            {#ix-attr:[Container(Layout.Stack)]}
            {#ix-attr:[Group(GroupLayout.GroupBox)]}
            {#ix-set:AttributeName = "<#Tool result 40#>"}
            ToolResult_40 : Axo_IV3_ToolResult;                                                     // IB852-IB871
            {#ix-attr:[Container(Layout.Stack)]}
            {#ix-attr:[Group(GroupLayout.GroupBox)]}
            {#ix-set:AttributeName = "<#Tool result 41#>"}
            ToolResult_41 : Axo_IV3_ToolResult;                                                     // IB872-IB891
            {#ix-attr:[Container(Layout.Stack)]}
            {#ix-attr:[Group(GroupLayout.GroupBox)]}
            {#ix-set:AttributeName = "<#Tool result 42#>"}
            ToolResult_42 : Axo_IV3_ToolResult;                                                     // IB892-IB911
            {#ix-attr:[Container(Layout.Stack)]}
            {#ix-attr:[Group(GroupLayout.GroupBox)]}
            {#ix-set:AttributeName = "<#Tool result 43#>"}
            ToolResult_43 : Axo_IV3_ToolResult;                                                     // IB912-IB931
            {#ix-attr:[Container(Layout.Stack)]}
            {#ix-attr:[Group(GroupLayout.GroupBox)]}
            {#ix-set:AttributeName = "<#Tool result 44#>"}
            ToolResult_44 : Axo_IV3_ToolResult;                                                     // IB932-IB951
            {#ix-attr:[Container(Layout.Stack)]}
            {#ix-attr:[Group(GroupLayout.GroupBox)]}
            {#ix-set:AttributeName = "<#Tool result 45#>"}
            ToolResult_45 : Axo_IV3_ToolResult;                                                     // IB952-IB971
            {#ix-attr:[Container(Layout.Stack)]}
            {#ix-attr:[Group(GroupLayout.GroupBox)]}
            {#ix-set:AttributeName = "<#Tool result 46#>"}
            ToolResult_46 : Axo_IV3_ToolResult;                                                     // IB972-IB991
            {#ix-attr:[Container(Layout.Stack)]}
            {#ix-attr:[Group(GroupLayout.GroupBox)]}
            {#ix-set:AttributeName = "<#Tool result 47#>"}
            ToolResult_47 : Axo_IV3_ToolResult;                                                     // IB992-IB1011
            {#ix-attr:[Container(Layout.Stack)]}
            {#ix-attr:[Group(GroupLayout.GroupBox)]}
            {#ix-set:AttributeName = "<#Tool result 48#>"}
            ToolResult_48 : Axo_IV3_ToolResult;                                                     // IB1012-IB1031
            {#ix-attr:[Container(Layout.Stack)]}
            {#ix-attr:[Group(GroupLayout.GroupBox)]}
            {#ix-set:AttributeName = "<#Tool result 49#>"}
            ToolResult_49 : Axo_IV3_ToolResult;                                                     // IB1032-IB1051
            {#ix-attr:[Container(Layout.Stack)]}
            {#ix-attr:[Group(GroupLayout.GroupBox)]}
            {#ix-set:AttributeName = "<#Tool result 50#>"}
            ToolResult_50 : Axo_IV3_ToolResult;                                                     // IB1052-IB1071
            {#ix-attr:[Container(Layout.Stack)]}
            {#ix-attr:[Group(GroupLayout.GroupBox)]}
            {#ix-set:AttributeName = "<#Tool result 51#>"}
            ToolResult_51 : Axo_IV3_ToolResult;                                                     // IB1072-IB1091
            {#ix-attr:[Container(Layout.Stack)]}
            {#ix-attr:[Group(GroupLayout.GroupBox)]}
            {#ix-set:AttributeName = "<#Tool result 52#>"}
            ToolResult_52 : Axo_IV3_ToolResult;                                                     // IB1092-IB1111
            {#ix-attr:[Container(Layout.Stack)]}
            {#ix-attr:[Group(GroupLayout.GroupBox)]}
            {#ix-set:AttributeName = "<#Tool result 53#>"}
            ToolResult_53 : Axo_IV3_ToolResult;                                                     // IB1112-IB1131
            {#ix-attr:[Container(Layout.Stack)]}
            {#ix-attr:[Group(GroupLayout.GroupBox)]}
            {#ix-set:AttributeName = "<#Tool result 54#>"}
            ToolResult_54 : Axo_IV3_ToolResult;                                                     // IB1132-IB1151
            {#ix-attr:[Container(Layout.Stack)]}
            {#ix-attr:[Group(GroupLayout.GroupBox)]}
            {#ix-set:AttributeName = "<#Tool result 55#>"}
            ToolResult_55 : Axo_IV3_ToolResult;                                                     // IB1152-IB1171
            {#ix-attr:[Container(Layout.Stack)]}
            {#ix-attr:[Group(GroupLayout.GroupBox)]}
            {#ix-set:AttributeName = "<#Tool result 56#>"}
            ToolResult_56 : Axo_IV3_ToolResult;                                                     // IB1172-IB1191
            {#ix-attr:[Container(Layout.Stack)]}
            {#ix-attr:[Group(GroupLayout.GroupBox)]}
            {#ix-set:AttributeName = "<#Tool result 57#>"}
            ToolResult_57 : Axo_IV3_ToolResult;                                                     // IB1192-IB1211
            {#ix-attr:[Container(Layout.Stack)]}
            {#ix-attr:[Group(GroupLayout.GroupBox)]}
            {#ix-set:AttributeName = "<#Tool result 58#>"}
            ToolResult_58 : Axo_IV3_ToolResult;                                                     // IB1212-IB1231
            {#ix-attr:[Container(Layout.Stack)]}
            {#ix-attr:[Group(GroupLayout.GroupBox)]}
            {#ix-set:AttributeName = "<#Tool result 59#>"}
            ToolResult_59 : Axo_IV3_ToolResult;                                                     // IB1232-IB1251
            {#ix-attr:[Container(Layout.Stack)]}
            {#ix-attr:[Group(GroupLayout.GroupBox)]}
            {#ix-set:AttributeName = "<#Tool result 60#>"}
            ToolResult_60 : Axo_IV3_ToolResult;                                                     // IB1252-IB1271
            {#ix-attr:[Container(Layout.Stack)]}
            {#ix-attr:[Group(GroupLayout.GroupBox)]}
            {#ix-set:AttributeName = "<#Tool result 61#>"}
            ToolResult_61 : Axo_IV3_ToolResult;                                                     // IB1272-IB1291
            {#ix-attr:[Container(Layout.Stack)]}
            {#ix-attr:[Group(GroupLayout.GroupBox)]}
            {#ix-set:AttributeName = "<#Tool result 62#>"}
            ToolResult_62 : Axo_IV3_ToolResult;                                                     // IB1292-IB1311
            {#ix-attr:[Container(Layout.Stack)]}
            {#ix-attr:[Group(GroupLayout.GroupBox)]}
            {#ix-set:AttributeName = "<#Tool result 63#>"}
            ToolResult_63 : Axo_IV3_ToolResult;                                                     // IB1312-IB1331
            {#ix-attr:[Container(Layout.Stack)]}
            {#ix-attr:[Group(GroupLayout.GroupBox)]}
            {#ix-set:AttributeName = "<#Tool result 64#>"}
            ToolResult_64 : Axo_IV3_ToolResult;                                                     // IB1332-IB1351

            {#ix-attr:[Container(Layout.Stack)]}
            {#ix-attr:[Group(GroupLayout.GroupBox)]}
            {#ix-set:AttributeName = "<#Device result bits 2#>"}
            {#ix-attr:[ReadOnly()]}
            DeviceResultBits_2          :   Axo_IV3_DeviceResultBits_2;                             // IB1352-IB1359

        END_VAR
    END_CLASS
END_NAMESPACE

(* ---- Axo_IV3_Out.st ---- *)
NAMESPACE AXOpen.Components.Keyence.Vision
    {S7.extern=ReadWrite}
    {#ix-attr:[Container(Layout.Wrap)]}
    CLASS PUBLIC Axo_IV3_Out
        VAR PUBLIC
            {#ix-set:AttributeName = "<#Command control#>"}
            {#ix-attr:[ReadOnly()]}
            CommandControl           :   Axo_IV3_CommandControl;
        END_VAR
    END_CLASS
END_NAMESPACE

(* ---- Axo_IV3_PositionAdjustResult.st ---- *)
NAMESPACE AXOpen.Components.Keyence.Vision
    {S7.extern=ReadWrite}
    {#ix-attr:[Container(Layout.Wrap)]}
    CLASS PUBLIC Axo_IV3_PositionAdjustResult
        VAR PUBLIC
            {#ix-attr:[Container(Layout.Stack)]}
            {#ix-attr:[Group(GroupLayout.GroupBox)]}
            {#ix-set:AttributeName = "<#Position correction score#>"}
            PositionCorrectionScore : UINT;                                                     // IW52
            {#ix-set:AttributeName = "<#Position correction score MAX#>"}
            PositionCorrectionScoreMAX : UINT;                                                  // IW54
            {#ix-set:AttributeName = "<#Position correction score MIN#>"}
            PositionCorrectionScoreMIN : UINT;                                                  // IW56
            {#ix-set:AttributeName = "<#Position correction score Lower threshold#>"}
            PositionCorrectionScoreLowerThreshold : UINT;                                       // IW58
                                                                                                // IB60-IB71
        END_VAR
    END_CLASS
END_NAMESPACE

(* ---- Axo_IV3_Status.st ---- *)
NAMESPACE AXOpen.Components.Keyence.Vision
    {S7.extern=ReadWrite}
    {#ix-attr:[Container(Layout.Stack)]}
    CLASS PUBLIC Axo_IV3_Status
        VAR PUBLIC

        END_VAR
    END_CLASS
END_NAMESPACE

(* ---- Axo_IV3_ToolResult.st ---- *)
NAMESPACE AXOpen.Components.Keyence.Vision
    {S7.extern=ReadWrite}
    {#ix-attr:[Container(Layout.Stack)]}
    CLASS PUBLIC Axo_IV3_ToolResult
        VAR PUBLIC
            {#ix-set:AttributeName = "<#Matching rate#>"}
            MatchingRate: UINT;
            {#ix-set:AttributeName = "<#Matching rate MAX#>"}
            MatchingRateMAX: UINT;
            {#ix-set:AttributeName = "<#Matching rate MIN#>"}
            MatchingRateMIN: UINT;
            {#ix-set:AttributeName = "<#Lower threshold#>"}
            LowerThreshold: UINT;
            {#ix-set:AttributeName = "<#Upper threshold#>"}
            UpperThreshold: UINT;
            {#ix-set:AttributeName = "<#Decimal point position#>"}
            DecimalPointPosition: UINT;
            {#ix-set:AttributeName = "<#Pitch present value MAX/color average H (hue)#>"}
            Data_1: UINT;
            {#ix-set:AttributeName = "<#Pitch present value MIN/color average S (saturation)#>"}
            Data_2: UINT;
            {#ix-set:AttributeName = "<#Number of pitches/color average V (brightness)/brightness average#>"}
            Data_3: UINT;
        END_VAR
    END_CLASS
END_NAMESPACE
